{attribute addProperty BoxType "EL7031-0000-0016"}
{attribute addProperty Id "StatusAT %I*Status_1C57BC2B162"}
{attribute addProperty CRC "3266366177"}
{attribute addProperty SizeInBites "16"}
{attribute addProperty SizeInBytes "2"}
TYPE STM_Status_C2B0CAE1 :
STRUCT
	{attribute addProperty Name "Status"}
	Status AT %I* : Status_1C57BC2B;
END_STRUCT
END_TYPE

(* stored: Version 1.2.0.0, ProductVersion 3.1.4024.9
   DUT STM_Status_C2B0CAE1: Id {899da4f6-ee76-40ab-afc1-6aefed13c91f} *)
